// TIA Portal project "function block1" (V16)

(* hardware
DEVICE "S7-1200 station_1"  S7-1200 Station
   slot 0: "Rack_0"  S7-1200 Rack  Rack  V1.0
   slot 1: "PLC_1"  CPU 1214C DC/DC/DC  6ES7 214-1AG40-0XB0  V4.4
   slot 2: "AI 4x13BIT/AQ 2x14BIT_1"  6ES7 234-4HE32-0XB0  V2.1
   slot 101: "CP 1243-7 LTE"  CP 1243-7 LTE  6GK7 243-7KX30-0XE0  V3.2
      slot 0: "Telecontrol server"  Partner
      slot 0: "Inter-station communication"  Partner
   slot 102: "RF120C_1"  RF120C  6GT2 002-0LA00  V1.0
   slot 103: "CM 1243-5"  CM 1243-5  6GK7 243-5DX30-0XE0  V1.3
*)

// ===== PLC "PLC_1"  CPU 1214C DC/DC/DC =====

VAR_GLOBAL   // PLC tag table "Default tag table"
   "switch" AT %M0.0 : Bool;
   "out" AT %M0.1 : Bool;
   "estop" AT %M0.2 : Bool;
   "esnotification" AT %M0.3 : Bool;
   "esalarm" AT %M0.4 : Bool;
   "alarmreset" AT %M0.5 : Bool;
   "alarmsilent" AT %M0.6 : Bool;
END_VAR

DATA_BLOCK "alarm_DB"   // DB1
{ S7_Optimized_Access := 'TRUE' }
VERSION : 0.1
// stored: InstanceOfName alarm
"alarm"
BEGIN
END_DATA_BLOCK

FUNCTION_BLOCK "alarm"   // FB1, LAD
{ S7_Optimized_Access := 'TRUE' }
VERSION : 0.1
   VAR
      ons : Bool;
      ons1 : Bool;
      ons2 : Bool;
      ons3 : Bool;
   END_VAR
   VAR_TEMP   // added for the SCL form of the ladder/FBD networks
      _w1 : Bool;
      _w2 : Bool;
      _w3 : Bool;
      _w4 : Bool;
   END_VAR
BEGIN

REGION Network 1
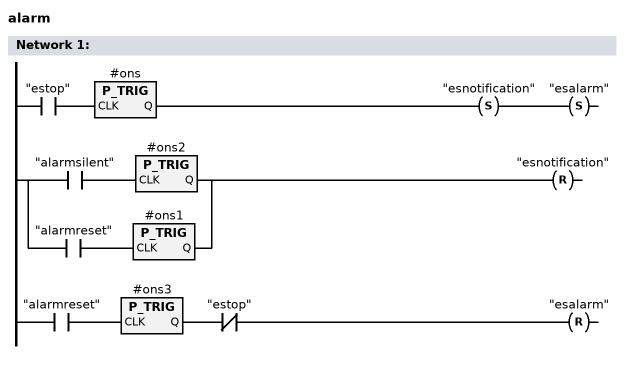
   RUNG wire#powerrail
      Contact( "estop" )
      P_Trig( #ons )
      S_Coil( "esnotification" )
      S_Coil( "esalarm" )
   END_RUNG
   RUNG wire#powerrail
      Contact( "alarmsilent" )
      P_Trig( #ons2 )
      wire#w1
      R_Coil( "esnotification" )
   END_RUNG
   RUNG wire#powerrail
      Contact( "alarmreset" )
      P_Trig( #ons1 )
   END_RUNG wire#w1
   RUNG wire#powerrail
      Contact( "alarmreset" )
      P_Trig( #ons3 )
      I_Contact( "estop" )
      R_Coil( "esalarm" )
   END_RUNG
   // the same network as SCL:
   #_w1 := "estop" AND NOT #ons;   // rising edge
   #ons := "estop";
   IF #_w1 THEN
       "esnotification" := TRUE;
       "esalarm" := TRUE;
   END_IF;
   #_w2 := "alarmsilent" AND NOT #ons2;   // rising edge
   #ons2 := "alarmsilent";
   #_w3 := "alarmreset" AND NOT #ons1;   // rising edge
   #ons1 := "alarmreset";
   IF #_w2 OR #_w3 THEN "esnotification" := FALSE; END_IF;
   #_w4 := "alarmreset" AND NOT #ons3;   // rising edge
   #ons3 := "alarmreset";
   IF #_w4 AND NOT "estop" THEN "esalarm" := FALSE; END_IF;
END_REGION
END_FUNCTION_BLOCK

ORGANIZATION_BLOCK "Main"   // OB1, LAD, ProgramCycle
TITLE = "Main Program Sweep (Cycle)"
{ S7_Optimized_Access := 'TRUE' }
VERSION : 0.1
   VAR_INPUT
      Initial_Call : Bool;   // Initial call of this OB
      Remanence : Bool;   // =True, if remanent data are available
   END_VAR
BEGIN

REGION Network 1
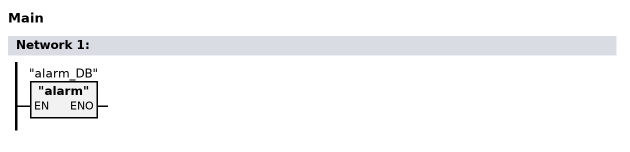
   RUNG wire#powerrail
      "alarm_DB"()
   END_RUNG
   // the same network as SCL:
   "alarm_DB"();   // "alarm"
END_REGION
END_ORGANIZATION_BLOCK